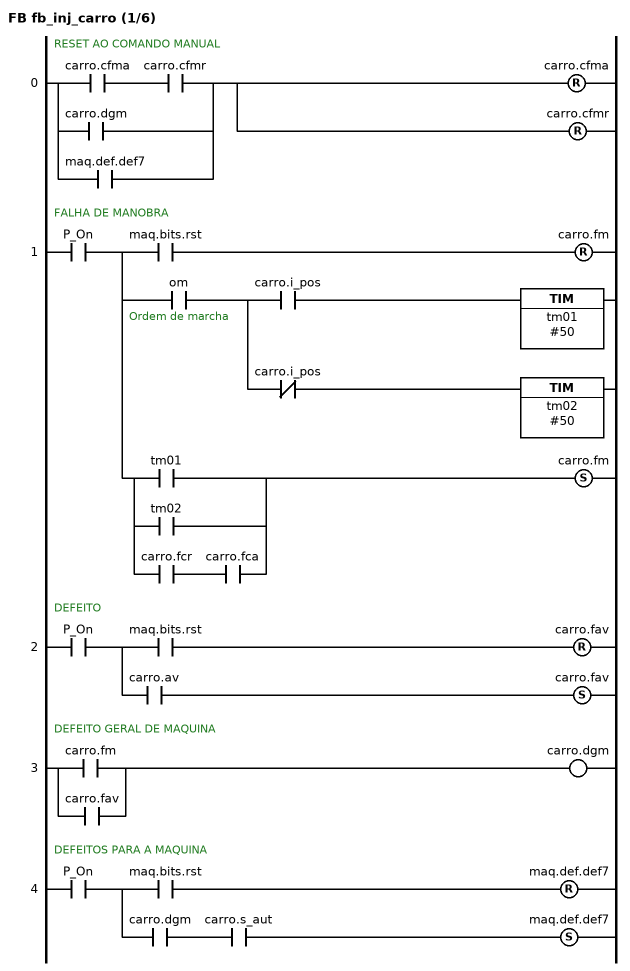
; [picture p48: FB fb_inj_carro, rungs 0-4]
; rung 0: RESET AO COMANDO MANUAL
LD carro.cfma
AND carro.cfmr
OR carro.dgm
OR maq.def.def7
RSET carro.cfma
RSET carro.cfmr
; rung 1: FALHA DE MANOBRA
LD P_On
OUT TR0
AND maq.bits.rst
RSET carro.fm
LD TR0
AND om  ; Ordem de marcha
OUT TR1
AND carro.i_pos
TIM tm01 #50
LD TR1
ANDNOT carro.i_pos
TIM tm02 #50
LD TR0
LD tm01
OR tm02
LD carro.fcr
AND carro.fca
ORLD
ANDLD
SET carro.fm
; rung 2: DEFEITO
LD P_On
OUT TR0
AND maq.bits.rst
RSET carro.fav
LD TR0
AND carro.av
SET carro.fav
; rung 3: DEFEITO GERAL DE MAQUINA
LD carro.fm
OR carro.fav
OUT carro.dgm
; rung 4: DEFEITOS PARA A MAQUINA
LD P_On
OUT TR0
AND maq.bits.rst
RSET maq.def.def7
LD TR0
AND carro.dgm
AND carro.s_aut
SET maq.def.def7

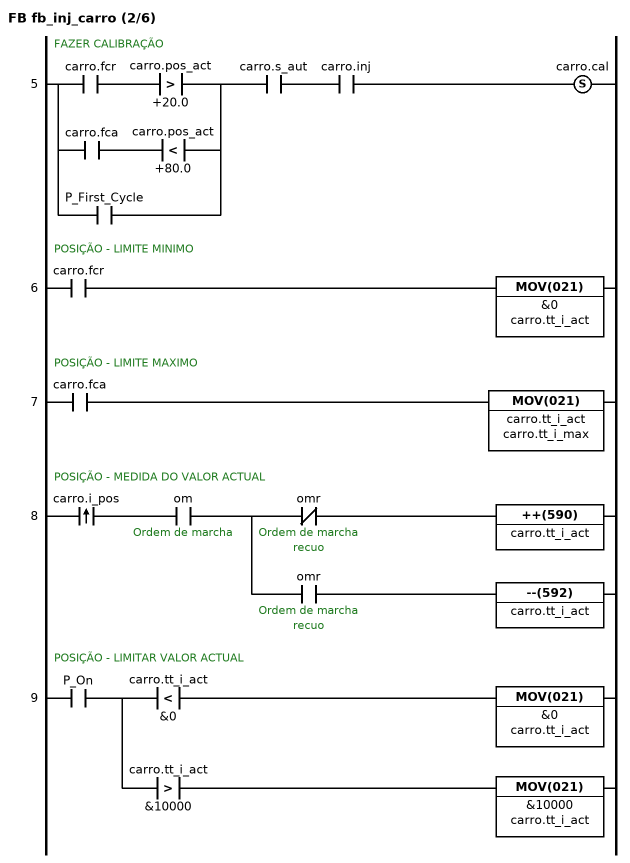
; rung 5: FAZER CALIBRAÇÃO
LD carro.fcr
AND>F(333) carro.pos_act +20.0
LD carro.fca
AND<F(331) carro.pos_act +80.0
ORLD
OR P_First_Cycle
AND carro.s_aut
AND carro.inj
SET carro.cal
; rung 6: POSIÇÃO - LIMITE MINIMO
LD carro.fcr
MOV(021) &0 carro.tt_i_act
; rung 7: POSIÇÃO - LIMITE MAXIMO
LD carro.fca
MOV(021) carro.tt_i_act carro.tt_i_max
; rung 8: POSIÇÃO - MEDIDA DO VALOR ACTUAL
@LD carro.i_pos
AND om  ; Ordem de marcha
OUT TR0
ANDNOT omr  ; Ordem de marcha recuo
++(590) carro.tt_i_act
LD TR0
AND omr  ; Ordem de marcha recuo
--(592) carro.tt_i_act
; rung 9: POSIÇÃO - LIMITAR VALOR ACTUAL
LD P_On
OUT TR0
AND<(310) carro.tt_i_act &0
MOV(021) &0 carro.tt_i_act
LD TR0
AND>(320) carro.tt_i_act &10000
MOV(021) &10000 carro.tt_i_act

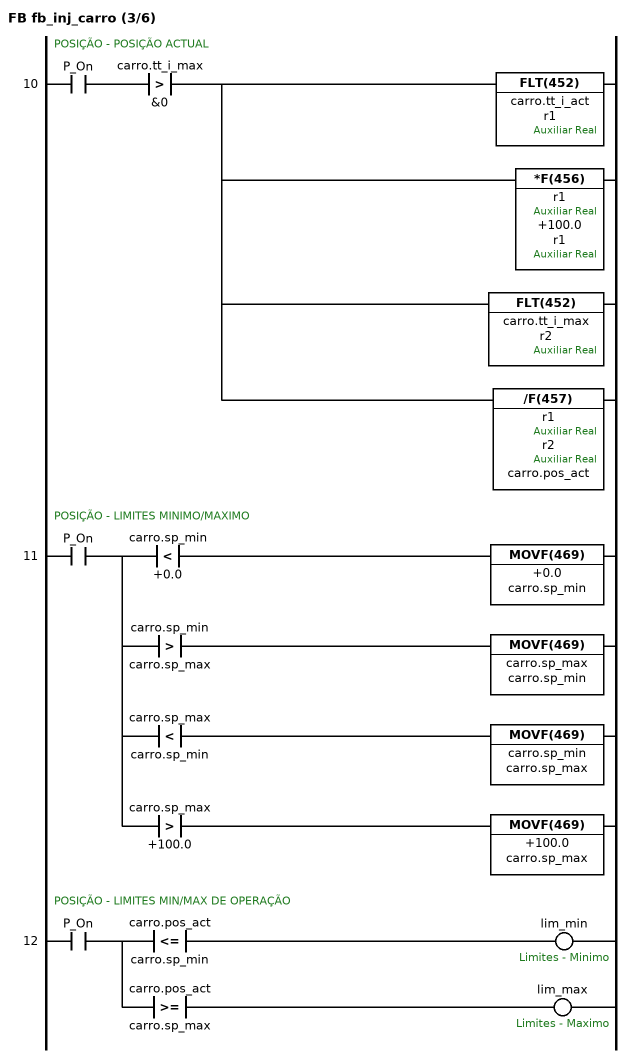
; rung 10: POSIÇÃO - POSIÇÃO ACTUAL
LD P_On
AND>(320) carro.tt_i_max &0
FLT(452) carro.tt_i_act r1  ; Auxiliar Real
*F(456) r1 +100.0 r1  ; Auxiliar Real
FLT(452) carro.tt_i_max r2  ; Auxiliar Real
/F(457) r1 r2 carro.pos_act  ; Auxiliar Real
; rung 11: POSIÇÃO - LIMITES MINIMO/MAXIMO
LD P_On
OUT TR0
AND<F(331) carro.sp_min +0.0
MOVF(469) +0.0 carro.sp_min
LD TR0
AND>F(333) carro.sp_min carro.sp_max
MOVF(469) carro.sp_max carro.sp_min
LD TR0
AND<F(331) carro.sp_max carro.sp_min
MOVF(469) carro.sp_min carro.sp_max
LD TR0
AND>F(333) carro.sp_max +100.0
MOVF(469) +100.0 carro.sp_max
; rung 12: POSIÇÃO - LIMITES MIN/MAX DE OPERAÇÃO
LD P_On
OUT TR0
AND<=F(332) carro.pos_act carro.sp_min
OUT lim_min  ; Limites - Minimo
LD TR0
AND>=F(334) carro.pos_act carro.sp_max
OUT lim_max  ; Limites - Maximo

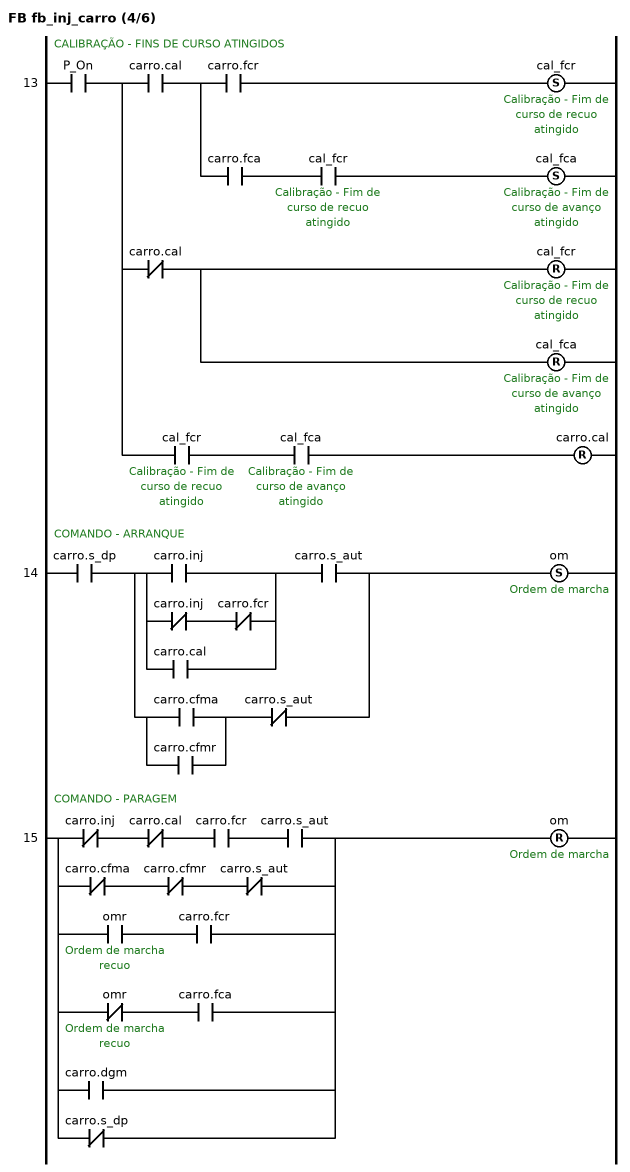
; rung 13: CALIBRAÇÃO - FINS DE CURSO ATINGIDOS
LD P_On
OUT TR0
AND carro.cal
OUT TR1
AND carro.fcr
SET cal_fcr  ; Calibração - Fim de curso de recuo atingido
LD TR1
AND carro.fca
AND cal_fcr  ; Calibração - Fim de curso de recuo atingido
SET cal_fca  ; Calibração - Fim de curso de avanço atingido
LD TR0
ANDNOT carro.cal
RSET cal_fcr  ; Calibração - Fim de curso de recuo atingido
RSET cal_fca  ; Calibração - Fim de curso de avanço atingido
LD TR0
AND cal_fcr  ; Calibração - Fim de curso de recuo atingido
AND cal_fca  ; Calibração - Fim de curso de avanço atingido
RSET carro.cal
; rung 14: COMANDO - ARRANQUE
LD carro.s_dp
LD carro.inj
LDNOT carro.inj
ANDNOT carro.fcr
ORLD
OR carro.cal
AND carro.s_aut
LD carro.cfma
OR carro.cfmr
ANDNOT carro.s_aut
ORLD
ANDLD
SET om  ; Ordem de marcha
; rung 15: COMANDO - PARAGEM
LDNOT carro.inj
ANDNOT carro.cal
AND carro.fcr
AND carro.s_aut
LDNOT carro.cfma
ANDNOT carro.cfmr
ANDNOT carro.s_aut
ORLD
LD omr  ; Ordem de marcha recuo
AND carro.fcr
ORLD
LDNOT omr  ; Ordem de marcha recuo
AND carro.fca
ORLD
OR carro.dgm
ORNOT carro.s_dp
RSET om  ; Ordem de marcha

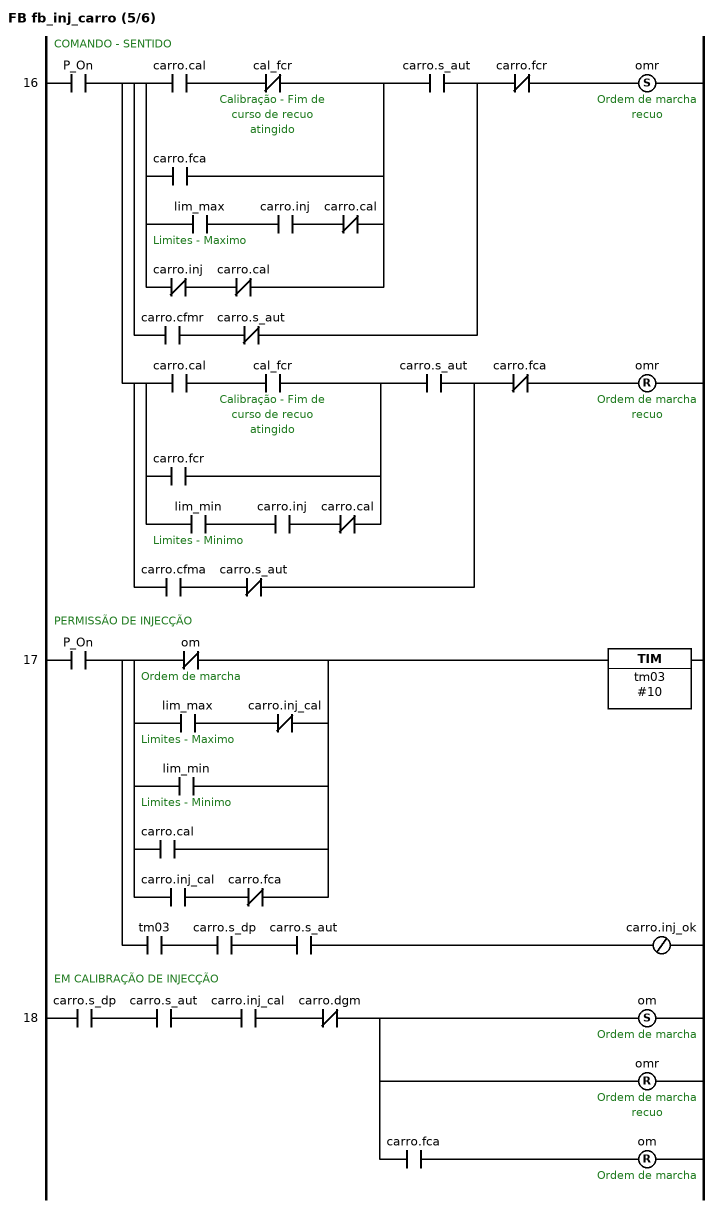
; rung 16: COMANDO - SENTIDO
LD P_On
OUT TR0
LD carro.cal
ANDNOT cal_fcr  ; Calibração - Fim de curso de recuo atingido
OR carro.fca
LD lim_max  ; Limites - Maximo
AND carro.inj
ANDNOT carro.cal
ORLD
LDNOT carro.inj
ANDNOT carro.cal
ORLD
AND carro.s_aut
LD carro.cfmr
ANDNOT carro.s_aut
ORLD
ANDLD
ANDNOT carro.fcr
SET omr  ; Ordem de marcha recuo
LD TR0
LD carro.cal
AND cal_fcr  ; Calibração - Fim de curso de recuo atingido
OR carro.fcr
LD lim_min  ; Limites - Minimo
AND carro.inj
ANDNOT carro.cal
ORLD
AND carro.s_aut
LD carro.cfma
ANDNOT carro.s_aut
ORLD
ANDLD
ANDNOT carro.fca
RSET omr  ; Ordem de marcha recuo
; rung 17: PERMISSÃO DE INJECÇÃO
LD P_On
OUT TR0
LDNOT om  ; Ordem de marcha
LD lim_max  ; Limites - Maximo
ANDNOT carro.inj_cal
ORLD
OR lim_min  ; Limites - Minimo
OR carro.cal
LD carro.inj_cal
ANDNOT carro.fca
ORLD
ANDLD
TIM tm03 #10
LD TR0
AND tm03
AND carro.s_dp
AND carro.s_aut
OUTNOT carro.inj_ok
; rung 18: EM CALIBRAÇÃO DE INJECÇÃO
LD carro.s_dp
AND carro.s_aut
AND carro.inj_cal
ANDNOT carro.dgm
SET om  ; Ordem de marcha
RSET omr  ; Ordem de marcha recuo
AND carro.fca
RSET om  ; Ordem de marcha

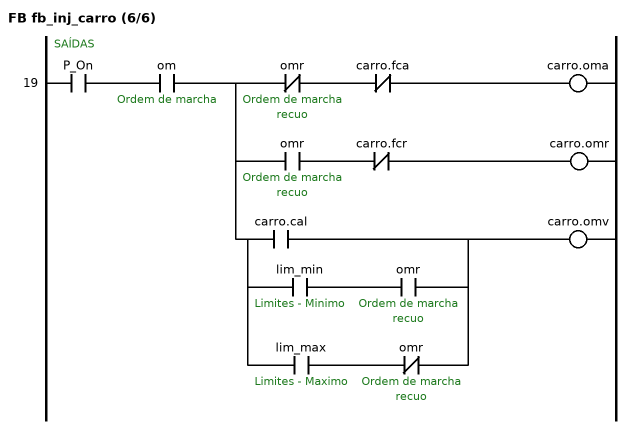
; rung 19: SAÍDAS
LD P_On
AND om  ; Ordem de marcha
OUT TR0
ANDNOT omr  ; Ordem de marcha recuo
ANDNOT carro.fca
OUT carro.oma
LD TR0
AND omr  ; Ordem de marcha recuo
ANDNOT carro.fcr
OUT carro.omr
LD TR0
LD carro.cal
LD lim_min  ; Limites - Minimo
AND omr  ; Ordem de marcha recuo
ORLD
LD lim_max  ; Limites - Maximo
ANDNOT omr  ; Ordem de marcha recuo
ORLD
ANDLD
OUT carro.omv

## Function block fb_inj_caudal
; FUNÇÃO CAUDALIMETRO - Caudalimetro local/remoto
VAR_IN_OUT
  tt : s_caudal;  (* Dados do caudalímetro *)
END_VAR
VAR
  tt_rem_d : REAL;  (* Diferença de totalização *)
  tm01 : TIMER;
  tm02 : TIMER;
  ct01 : COUNTER;
END_VAR

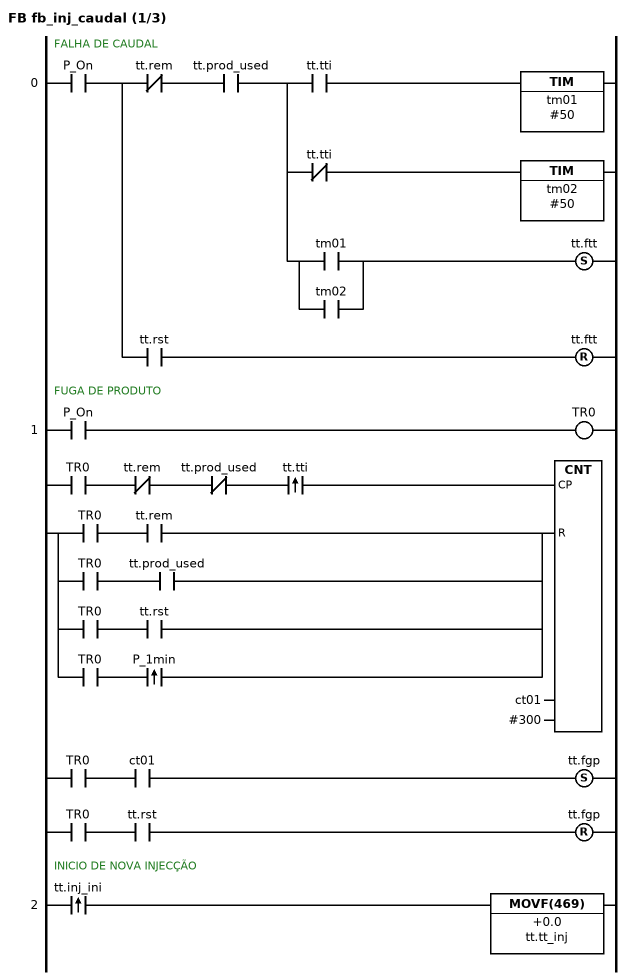
; rung 0: FALHA DE CAUDAL
LD P_On
OUT TR0
ANDNOT tt.rem
AND tt.prod_used
OUT TR1
AND tt.tti
TIM tm01 #50
LD TR1
ANDNOT tt.tti
TIM tm02 #50
LD TR1
LD tm01
OR tm02
ANDLD
SET tt.ftt
LD TR0
AND tt.rst
RSET tt.ftt
; rung 1: FUGA DE PRODUTO
LD P_On
OUT TR0
LD TR0
ANDNOT tt.rem
ANDNOT tt.prod_used
@AND tt.tti
LD TR0
AND tt.rem
LD TR0
AND tt.prod_used
ORLD
LD TR0
AND tt.rst
ORLD
LD TR0
@AND P_1min
ORLD
CNT ct01 #300
LD TR0
AND ct01
SET tt.fgp
LD TR0
AND tt.rst
RSET tt.fgp
; rung 2: INICIO DE NOVA INJECÇÃO
@LD tt.inj_ini
MOVF(469) +0.0 tt.tt_inj

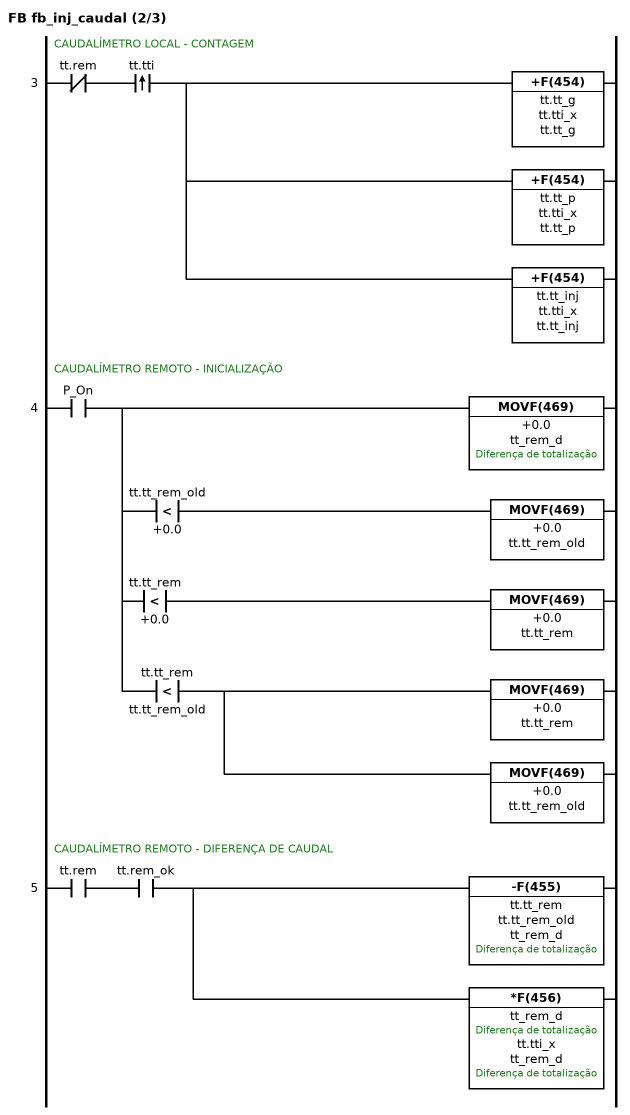
; rung 3: CAUDALÍMETRO LOCAL - CONTAGEM
LDNOT tt.rem
@AND tt.tti
+F(454) tt.tt_g tt.tti_x tt.tt_g
+F(454) tt.tt_p tt.tti_x tt.tt_p
+F(454) tt.tt_inj tt.tti_x tt.tt_inj
; rung 4: CAUDALÍMETRO REMOTO - INICIALIZAÇÃO
LD P_On
OUT TR0
MOVF(469) +0.0 tt_rem_d  ; Diferença de totalização
AND<F(331) tt.tt_rem_old +0.0
MOVF(469) +0.0 tt.tt_rem_old
LD TR0
AND<F(331) tt.tt_rem +0.0
MOVF(469) +0.0 tt.tt_rem
LD TR0
AND<F(331) tt.tt_rem tt.tt_rem_old
MOVF(469) +0.0 tt.tt_rem
MOVF(469) +0.0 tt.tt_rem_old
; rung 5: CAUDALÍMETRO REMOTO - DIFERENÇA DE CAUDAL
LD tt.rem
AND tt.rem_ok
-F(455) tt.tt_rem tt.tt_rem_old tt_rem_d  ; Diferença de totalização
*F(456) tt_rem_d tt.tti_x tt_rem_d  ; Diferença de totalização

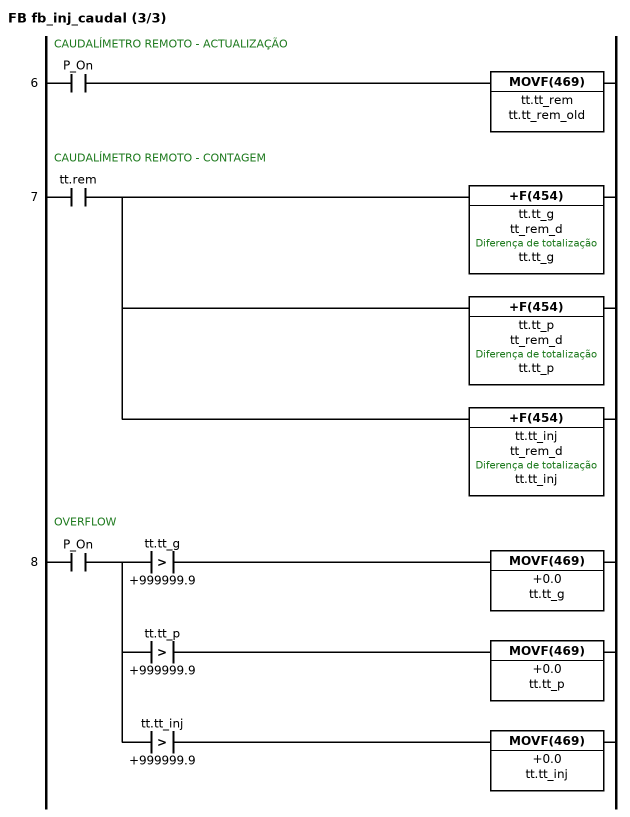
; rung 6: CAUDALÍMETRO REMOTO - ACTUALIZAÇÃO
LD P_On
MOVF(469) tt.tt_rem tt.tt_rem_old
; rung 7: CAUDALÍMETRO REMOTO - CONTAGEM
LD tt.rem
+F(454) tt.tt_g tt_rem_d tt.tt_g  ; Diferença de totalização
+F(454) tt.tt_p tt_rem_d tt.tt_p  ; Diferença de totalização
+F(454) tt.tt_inj tt_rem_d tt.tt_inj  ; Diferença de totalização
; rung 8: OVERFLOW
LD P_On
OUT TR0
AND>F(333) tt.tt_g +999999.9
MOVF(469) +0.0 tt.tt_g
LD TR0
AND>F(333) tt.tt_p +999999.9
MOVF(469) +0.0 tt.tt_p
LD TR0
AND>F(333) tt.tt_inj +999999.9
MOVF(469) +0.0 tt.tt_inj

## Function block fb_maquina
; FUNÇÃO MAQUINA - Faz a gestão dos passos e comandos aos vários blocos.
VAR_INPUT
  Rcp_OK : BOOL;
END_VAR
VAR_IN_OUT
  maq : s_maquina;  (* Dados da maquina *)
  of1_exe : s_of;  (* Dados da OF a ser executada *)
  of2_maq : s_of;  (* Dados da OF carregados na maquina *)
  of3_trp : s_of;  (* Dados da OF recebidos do transporte *)
  mes_com : s_mes_com;  (* Dados da comunição com o MES *)
  prg_exe : s_of_prg;  (* Programa a executar *)
  prg_on : s_of_prg;  (* Programa online *)
  Estado : s_Estado;
  F_Ciclo_bit : BOOL;
END_VAR
VAR
  fb_maquina_mov_pss_act : fb_maquina_mov_pss_act;
  fb_of_copy : fb_of_copy;
  fb_of_clear : fb_of_clear;
  fb_mes_com_exe : fb_mes_com_exe;
  fb_maquina_copy_log : fb_maquina_copy_log;
  fb_of_copy_of_prg_prg : fb_of_copy_of_prg_prg;
  fb_of_exe_calc : fb_of_exe_calc;
  log_tipo : INT;  (* Tipo de copia: 0 - Copia user/lote e dados a zero / 1 - Copia com ordem a decorrer (não copia user/lote) / 2 - Fim da ordem (Coloca passo 999) / 3 - Ordem descarregada sem execução (Colocar -3 no passo) *)
  tm01 : TIMER;
  tm02 : TIMER;
  tm03 : TIMER;
  tm04 : TIMER;
  tm05 : TIMER;
  tm06 : TIMER;
  tm07 : TIMER;
  tm08 : TIMER;
  tm09 : TIMER;
  tm10 : TIMER;
  tm11 : TIMER;
  tm12 : TIMER;
  tm13 : TIMER;
  tm14 : TIMER;
  tm15 : TIMER;
  tm16 : TIMER;
  of_trat : BOOL;  (* Ordem tratada *)
END_VAR

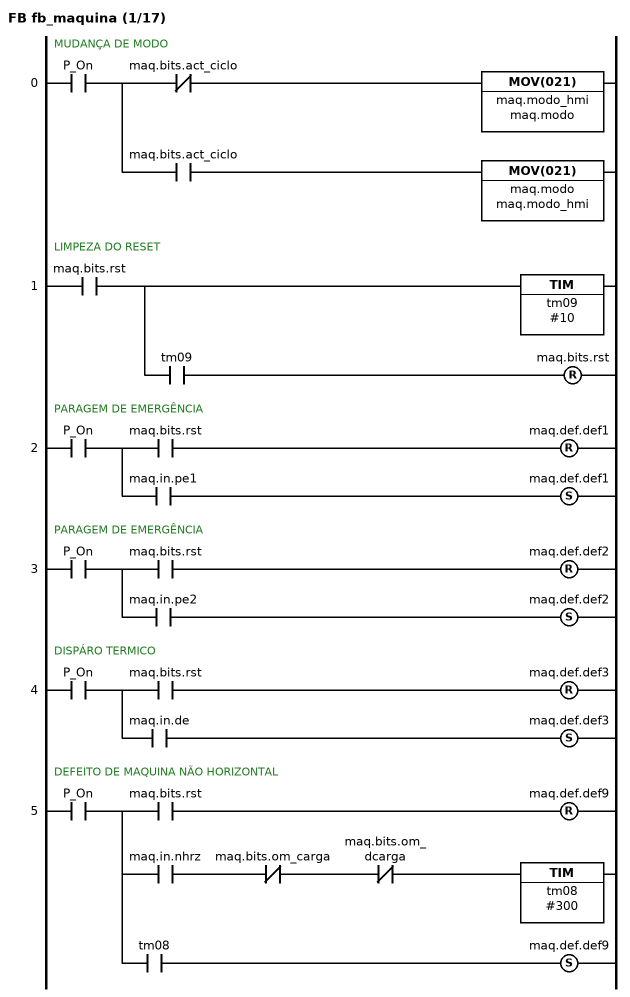
; rung 0: MUDANÇA DE MODO
LD P_On
OUT TR0
ANDNOT maq.bits.act_ciclo
MOV(021) maq.modo_hmi maq.modo
LD TR0
AND maq.bits.act_ciclo
MOV(021) maq.modo maq.modo_hmi
; rung 1: LIMPEZA DO RESET
LD maq.bits.rst
TIM tm09 #10
AND tm09
RSET maq.bits.rst
; rung 2: PARAGEM DE EMERGÊNCIA
LD P_On
OUT TR0
AND maq.bits.rst
RSET maq.def.def1
LD TR0
AND maq.in.pe1
SET maq.def.def1
; rung 3: PARAGEM DE EMERGÊNCIA
LD P_On
OUT TR0
AND maq.bits.rst
RSET maq.def.def2
LD TR0
AND maq.in.pe2
SET maq.def.def2
; rung 4: DISPÁRO TERMICO
LD P_On
OUT TR0
AND maq.bits.rst
RSET maq.def.def3
LD TR0
AND maq.in.de
SET maq.def.def3
; rung 5: DEFEITO DE MAQUINA NÃO HORIZONTAL
LD P_On
OUT TR0
AND maq.bits.rst
RSET maq.def.def9
LD TR0
AND maq.in.nhrz
ANDNOT maq.bits.om_carga
ANDNOT maq.bits.om_dcarga
TIM tm08 #300
LD TR0
AND tm08
SET maq.def.def9

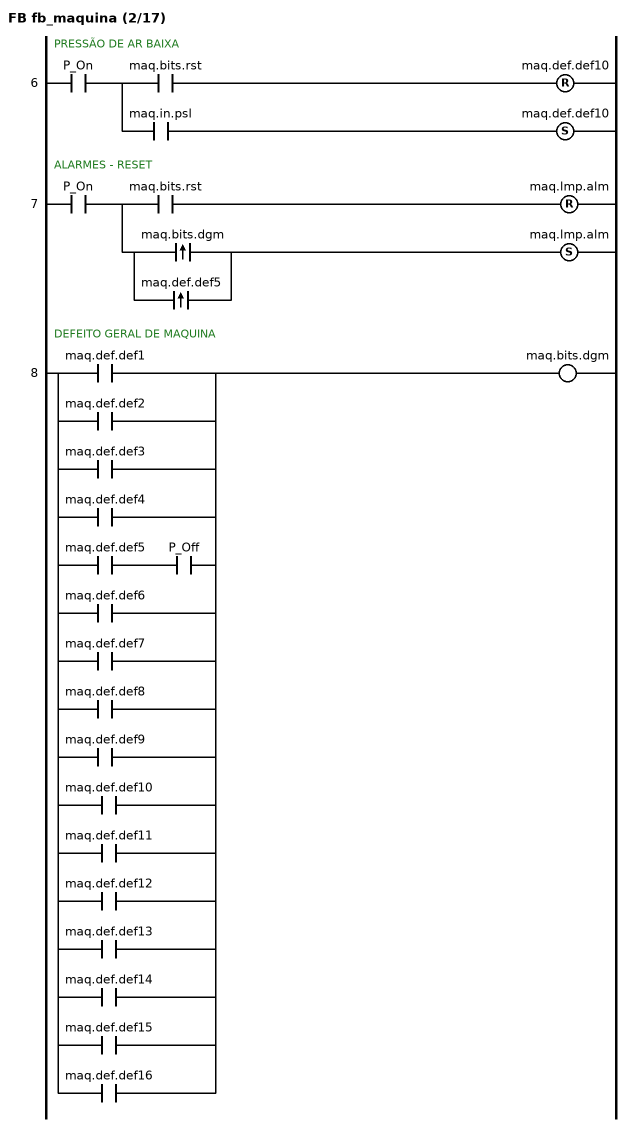
; rung 6: PRESSÃO DE AR BAIXA
LD P_On
OUT TR0
AND maq.bits.rst
RSET maq.def.def10
LD TR0
AND maq.in.psl
SET maq.def.def10
; rung 7: ALARMES - RESET
LD P_On
OUT TR0
AND maq.bits.rst
RSET maq.lmp.alm
LD TR0
@LD maq.bits.dgm
@OR maq.def.def5
ANDLD
SET maq.lmp.alm
; rung 8: DEFEITO GERAL DE MAQUINA
LD maq.def.def1
OR maq.def.def2
OR maq.def.def3
OR maq.def.def4
LD maq.def.def5
AND P_Off
ORLD
OR maq.def.def6
OR maq.def.def7
OR maq.def.def8
OR maq.def.def9
OR maq.def.def10
OR maq.def.def11
OR maq.def.def12
OR maq.def.def13
OR maq.def.def14
OR maq.def.def15
OR maq.def.def16
OUT maq.bits.dgm

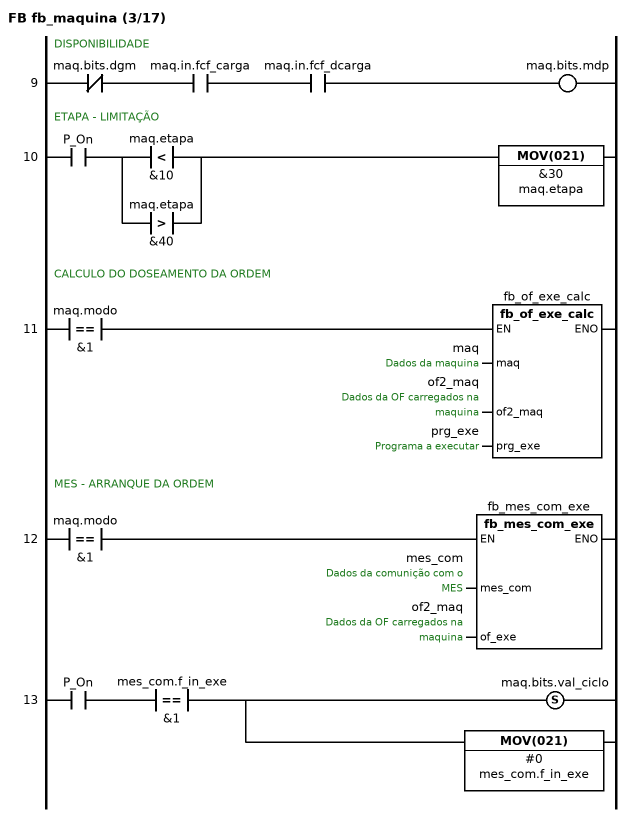
; rung 9: DISPONIBILIDADE
LDNOT maq.bits.dgm
AND maq.in.fcf_carga
AND maq.in.fcf_dcarga
OUT maq.bits.mdp
; rung 10: ETAPA - LIMITAÇÃO
LD P_On
LD<(310) maq.etapa &10
OR>(320) maq.etapa &40
ANDLD
MOV(021) &30 maq.etapa
; rung 11: CALCULO DO DOSEAMENTO DA ORDEM
LD=(300) maq.modo &1
CALL fb_of_exe_calc : fb_of_exe_calc (maq := maq, of2_maq := of2_maq, prg_exe := prg_exe)  ; Dados da maquina, Dados da OF carregados na maquina, Programa a executar
; rung 12: MES - ARRANQUE DA ORDEM
LD=(300) maq.modo &1
CALL fb_mes_com_exe : fb_mes_com_exe (mes_com := mes_com, of_exe := of2_maq)  ; Dados da comunição com o MES, Dados da OF carregados na maquina
; rung 13
LD P_On
AND=(300) mes_com.f_in_exe &1
SET maq.bits.val_ciclo
MOV(021) #0 mes_com.f_in_exe

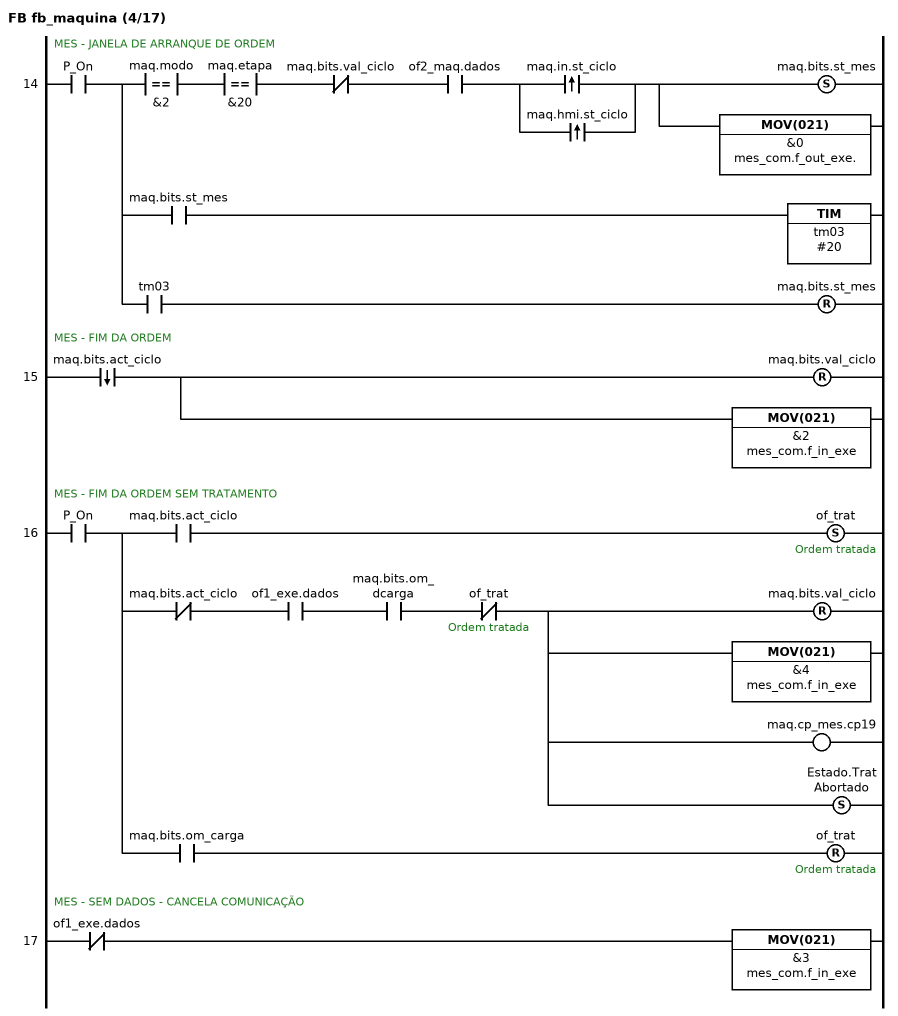
; rung 14: MES - JANELA DE ARRANQUE DE ORDEM
LD P_On
OUT TR0
AND=(300) maq.modo &2
AND=(300) maq.etapa &20
ANDNOT maq.bits.val_ciclo
AND of2_maq.dados
@LD maq.in.st_ciclo
@OR maq.hmi.st_ciclo
ANDLD
SET maq.bits.st_mes
MOV(021) &0 mes_com.f_out_exe.
LD TR0
AND maq.bits.st_mes
TIM tm03 #20
LD TR0
AND tm03
RSET maq.bits.st_mes
; rung 15: MES - FIM DA ORDEM
%LD maq.bits.act_ciclo
RSET maq.bits.val_ciclo
MOV(021) &2 mes_com.f_in_exe
; rung 16: MES - FIM DA ORDEM SEM TRATAMENTO
LD P_On
OUT TR0
AND maq.bits.act_ciclo
SET of_trat  ; Ordem tratada
LD TR0
ANDNOT maq.bits.act_ciclo
AND of1_exe.dados
AND maq.bits.om_dcarga
ANDNOT of_trat  ; Ordem tratada
RSET maq.bits.val_ciclo
MOV(021) &4 mes_com.f_in_exe
OUT maq.cp_mes.cp19
SET Estado.TratAbortado
LD TR0
AND maq.bits.om_carga
RSET of_trat  ; Ordem tratada
; rung 17: MES - SEM DADOS - CANCELA COMUNICAÇÃO
LDNOT of1_exe.dados
MOV(021) &3 mes_com.f_in_exe

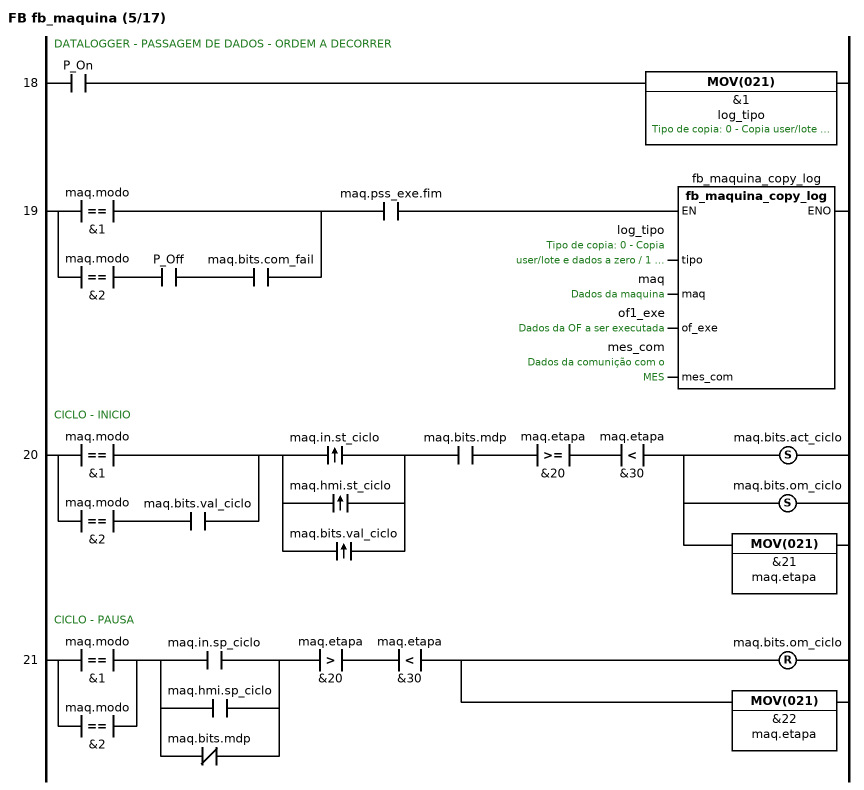
; rung 18: DATALOGGER - PASSAGEM DE DADOS - ORDEM A DECORRER
LD P_On
MOV(021) &1 log_tipo  ; Tipo de copia: 0 - Copia user/lote e dados a zero / 1 - Copia com ordem a decorrer (não copia user/lote) / 2 - Fim da ordem (Coloca passo 999) / 3 - Ordem descarregada sem execução (Colocar -3 no passo)
; rung 19
LD=(300) maq.modo &1
LD=(300) maq.modo &2
AND P_Off
AND maq.bits.com_fail
ORLD
AND maq.pss_exe.fim
CALL fb_maquina_copy_log : fb_maquina_copy_log (tipo := log_tipo, maq := maq, of_exe := of1_exe, mes_com := mes_com)  ; Tipo de copia: 0 - Copia user/lote e dados a zero / 1 - Copia com ordem a decorrer (não copia user/lote) / 2 - Fim da ordem (Coloca passo 999) / 3 - Ordem descarregada sem execução (Colocar -3 no passo), Dados da maquina, Dados da OF a ser executada, Dados da comunição com o MES
; rung 20: CICLO - INICIO
LD=(300) maq.modo &1
LD=(300) maq.modo &2
AND maq.bits.val_ciclo
ORLD
@LD maq.in.st_ciclo
@OR maq.hmi.st_ciclo
@OR maq.bits.val_ciclo
ANDLD
AND maq.bits.mdp
AND>=(325) maq.etapa &20
AND<(310) maq.etapa &30
SET maq.bits.act_ciclo
SET maq.bits.om_ciclo
MOV(021) &21 maq.etapa
; rung 21: CICLO - PAUSA
LD=(300) maq.modo &1
OR=(300) maq.modo &2
LD maq.in.sp_ciclo
OR maq.hmi.sp_ciclo
ORNOT maq.bits.mdp
ANDLD
AND>(320) maq.etapa &20
AND<(310) maq.etapa &30
RSET maq.bits.om_ciclo
MOV(021) &22 maq.etapa

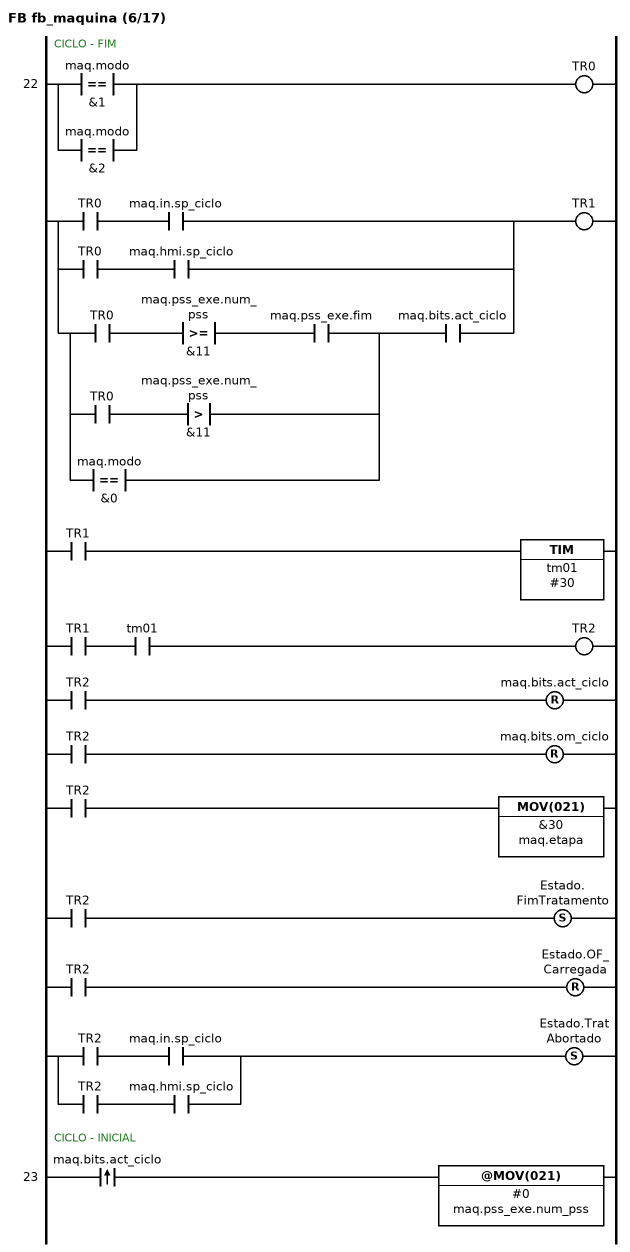
; rung 22: CICLO - FIM
LD=(300) maq.modo &1
OR=(300) maq.modo &2
OUT TR0
LD TR0
AND maq.in.sp_ciclo
LD TR0
AND maq.hmi.sp_ciclo
ORLD
LD TR0
AND>=(325) maq.pss_exe.num_pss &11
AND maq.pss_exe.fim
LD TR0
AND>(320) maq.pss_exe.num_pss &11
ORLD
OR=(300) maq.modo &0
AND maq.bits.act_ciclo
ORLD
OUT TR1
LD TR1
TIM tm01 #30
LD TR1
AND tm01
OUT TR2
LD TR2
RSET maq.bits.act_ciclo
LD TR2
RSET maq.bits.om_ciclo
LD TR2
MOV(021) &30 maq.etapa
LD TR2
SET Estado.FimTratamento
LD TR2
RSET Estado.OF_Carregada
LD TR2
AND maq.in.sp_ciclo
LD TR2
AND maq.hmi.sp_ciclo
ORLD
SET Estado.TratAbortado
; rung 23: CICLO - INICIAL
@LD maq.bits.act_ciclo
@MOV(021) #0 maq.pss_exe.num_pss

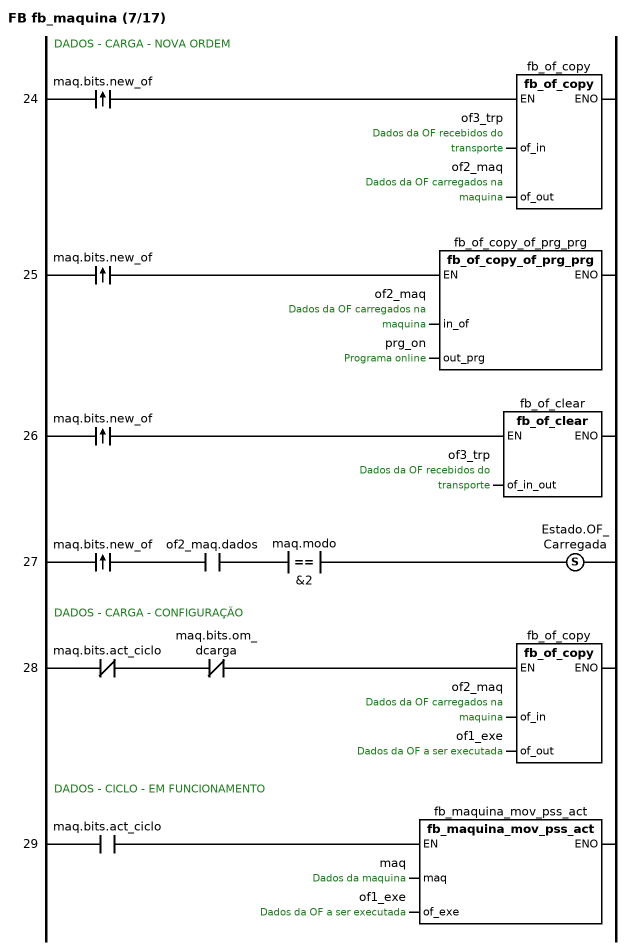
; rung 24: DADOS - CARGA - NOVA ORDEM
@LD maq.bits.new_of
CALL fb_of_copy : fb_of_copy (of_in := of3_trp, of_out := of2_maq)  ; Dados da OF recebidos do transporte, Dados da OF carregados na maquina
; rung 25
@LD maq.bits.new_of
CALL fb_of_copy_of_prg_prg : fb_of_copy_of_prg_prg (in_of := of2_maq, out_prg := prg_on)  ; Dados da OF carregados na maquina, Programa online
; rung 26
@LD maq.bits.new_of
CALL fb_of_clear : fb_of_clear (of_in_out := of3_trp)  ; Dados da OF recebidos do transporte
; rung 27
@LD maq.bits.new_of
AND of2_maq.dados
AND=(300) maq.modo &2
SET Estado.OF_Carregada
; rung 28: DADOS - CARGA - CONFIGURAÇÃO
LDNOT maq.bits.act_ciclo
ANDNOT maq.bits.om_dcarga
CALL fb_of_copy : fb_of_copy (of_in := of2_maq, of_out := of1_exe)  ; Dados da OF carregados na maquina, Dados da OF a ser executada
; rung 29: DADOS - CICLO - EM FUNCIONAMENTO
LD maq.bits.act_ciclo
CALL fb_maquina_mov_pss_act : fb_maquina_mov_pss_act (maq := maq, of_exe := of1_exe)  ; Dados da maquina, Dados da OF a ser executada

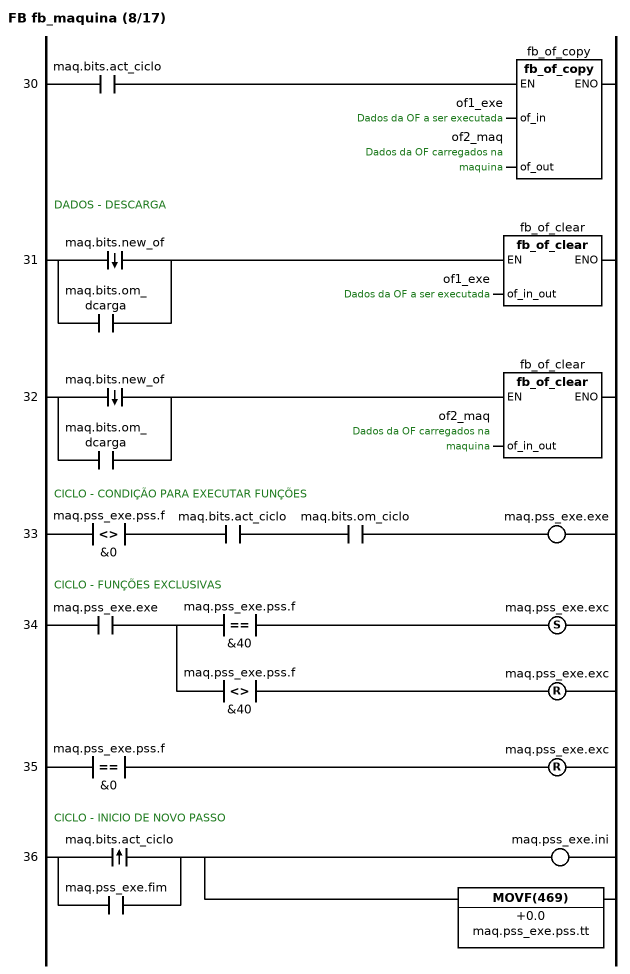
; rung 30
LD maq.bits.act_ciclo
CALL fb_of_copy : fb_of_copy (of_in := of1_exe, of_out := of2_maq)  ; Dados da OF a ser executada, Dados da OF carregados na maquina
; rung 31: DADOS - DESCARGA
%LD maq.bits.new_of
OR maq.bits.om_dcarga
CALL fb_of_clear : fb_of_clear (of_in_out := of1_exe)  ; Dados da OF a ser executada
; rung 32
%LD maq.bits.new_of
OR maq.bits.om_dcarga
CALL fb_of_clear : fb_of_clear (of_in_out := of2_maq)  ; Dados da OF carregados na maquina
; rung 33: CICLO - CONDIÇÃO PARA EXECUTAR FUNÇÕES
LD<>(305) maq.pss_exe.pss.f &0
AND maq.bits.act_ciclo
AND maq.bits.om_ciclo
OUT maq.pss_exe.exe
; rung 34: CICLO - FUNÇÕES EXCLUSIVAS
LD maq.pss_exe.exe
OUT TR0
AND=(300) maq.pss_exe.pss.f &40
SET maq.pss_exe.exc
LD TR0
AND<>(305) maq.pss_exe.pss.f &40
RSET maq.pss_exe.exc
; rung 35
LD=(300) maq.pss_exe.pss.f &0
RSET maq.pss_exe.exc
; rung 36: CICLO - INICIO DE NOVO PASSO
@LD maq.bits.act_ciclo
OR maq.pss_exe.fim
OUT maq.pss_exe.ini
MOVF(469) +0.0 maq.pss_exe.pss.tt

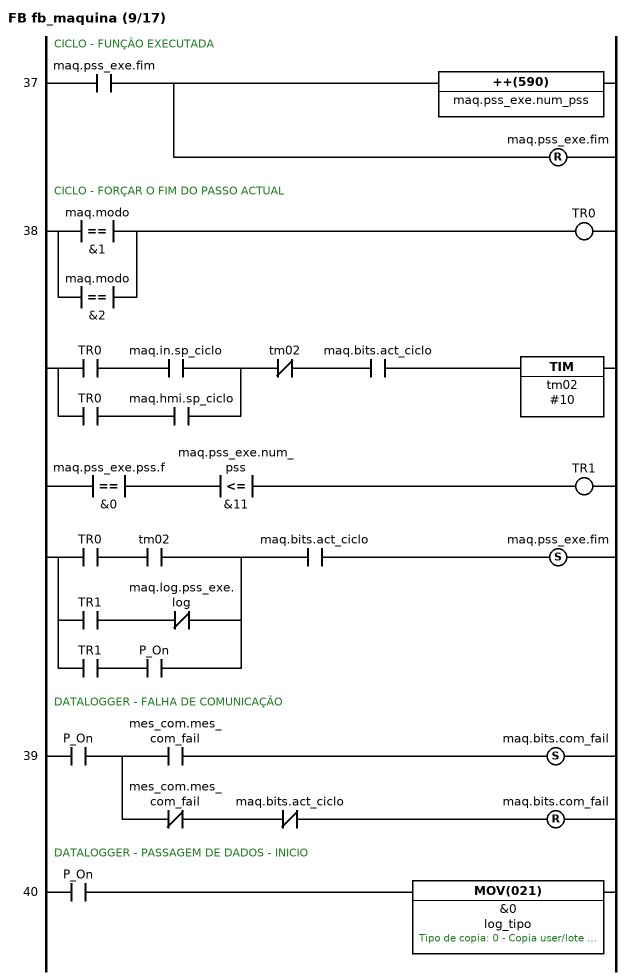
; rung 37: CICLO - FUNÇÃO EXECUTADA
LD maq.pss_exe.fim
++(590) maq.pss_exe.num_pss
RSET maq.pss_exe.fim
; rung 38: CICLO - FORÇAR O FIM DO PASSO ACTUAL
LD=(300) maq.modo &1
OR=(300) maq.modo &2
OUT TR0
LD TR0
AND maq.in.sp_ciclo
LD TR0
AND maq.hmi.sp_ciclo
ORLD
ANDNOT tm02
AND maq.bits.act_ciclo
TIM tm02 #10
LD=(300) maq.pss_exe.pss.f &0
AND<=(315) maq.pss_exe.num_pss &11
OUT TR1
LD TR0
AND tm02
LD TR1
ANDNOT maq.log.pss_exe.log
ORLD
LD TR1
AND P_On
ORLD
AND maq.bits.act_ciclo
SET maq.pss_exe.fim
; rung 39: DATALOGGER - FALHA DE COMUNICAÇÃO
LD P_On
OUT TR0
AND mes_com.mes_com_fail
SET maq.bits.com_fail
LD TR0
ANDNOT mes_com.mes_com_fail
ANDNOT maq.bits.act_ciclo
RSET maq.bits.com_fail
; rung 40: DATALOGGER - PASSAGEM DE DADOS - INICIO
LD P_On
MOV(021) &0 log_tipo  ; Tipo de copia: 0 - Copia user/lote e dados a zero / 1 - Copia com ordem a decorrer (não copia user/lote) / 2 - Fim da ordem (Coloca passo 999) / 3 - Ordem descarregada sem execução (Colocar -3 no passo)

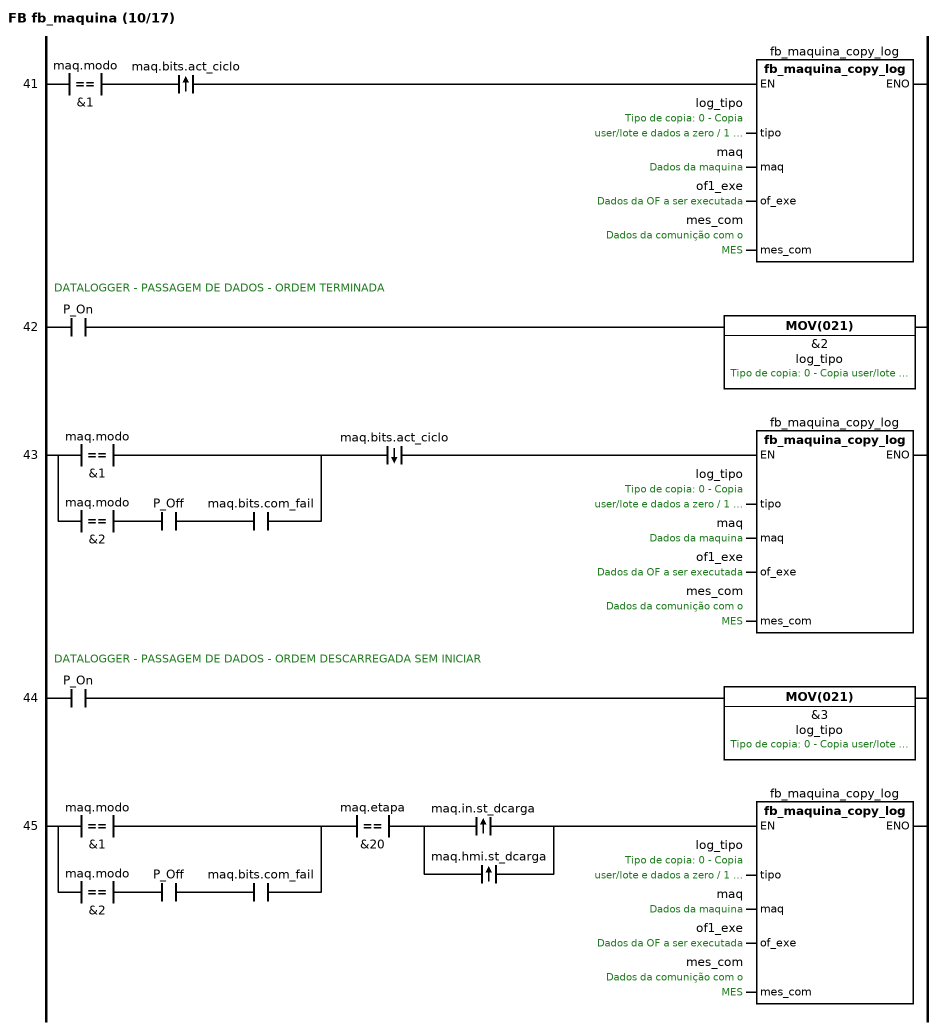
; rung 41
LD=(300) maq.modo &1
@AND maq.bits.act_ciclo
CALL fb_maquina_copy_log : fb_maquina_copy_log (tipo := log_tipo, maq := maq, of_exe := of1_exe, mes_com := mes_com)  ; Tipo de copia: 0 - Copia user/lote e dados a zero / 1 - Copia com ordem a decorrer (não copia user/lote) / 2 - Fim da ordem (Coloca passo 999) / 3 - Ordem descarregada sem execução (Colocar -3 no passo), Dados da maquina, Dados da OF a ser executada, Dados da comunição com o MES
; rung 42: DATALOGGER - PASSAGEM DE DADOS - ORDEM TERMINADA
LD P_On
MOV(021) &2 log_tipo  ; Tipo de copia: 0 - Copia user/lote e dados a zero / 1 - Copia com ordem a decorrer (não copia user/lote) / 2 - Fim da ordem (Coloca passo 999) / 3 - Ordem descarregada sem execução (Colocar -3 no passo)
; rung 43
LD=(300) maq.modo &1
LD=(300) maq.modo &2
AND P_Off
AND maq.bits.com_fail
ORLD
%AND maq.bits.act_ciclo
CALL fb_maquina_copy_log : fb_maquina_copy_log (tipo := log_tipo, maq := maq, of_exe := of1_exe, mes_com := mes_com)  ; Tipo de copia: 0 - Copia user/lote e dados a zero / 1 - Copia com ordem a decorrer (não copia user/lote) / 2 - Fim da ordem (Coloca passo 999) / 3 - Ordem descarregada sem execução (Colocar -3 no passo), Dados da maquina, Dados da OF a ser executada, Dados da comunição com o MES
; rung 44: DATALOGGER - PASSAGEM DE DADOS - ORDEM DESCARREGADA SEM INICIAR
LD P_On
MOV(021) &3 log_tipo  ; Tipo de copia: 0 - Copia user/lote e dados a zero / 1 - Copia com ordem a decorrer (não copia user/lote) / 2 - Fim da ordem (Coloca passo 999) / 3 - Ordem descarregada sem execução (Colocar -3 no passo)
; rung 45
LD=(300) maq.modo &1
LD=(300) maq.modo &2
AND P_Off
AND maq.bits.com_fail
ORLD
AND=(300) maq.etapa &20
@LD maq.in.st_dcarga
@OR maq.hmi.st_dcarga
ANDLD
CALL fb_maquina_copy_log : fb_maquina_copy_log (tipo := log_tipo, maq := maq, of_exe := of1_exe, mes_com := mes_com)  ; Tipo de copia: 0 - Copia user/lote e dados a zero / 1 - Copia com ordem a decorrer (não copia user/lote) / 2 - Fim da ordem (Coloca passo 999) / 3 - Ordem descarregada sem execução (Colocar -3 no passo), Dados da maquina, Dados da OF a ser executada, Dados da comunição com o MES

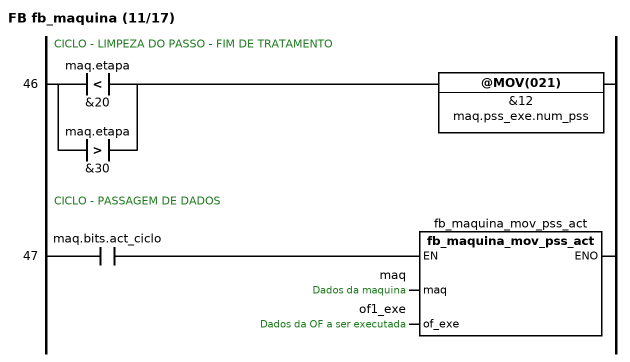
; rung 46: CICLO - LIMPEZA DO PASSO - FIM DE TRATAMENTO
LD<(310) maq.etapa &20
OR>(320) maq.etapa &30
@MOV(021) &12 maq.pss_exe.num_pss
; rung 47: CICLO - PASSAGEM DE DADOS
LD maq.bits.act_ciclo
CALL fb_maquina_mov_pss_act : fb_maquina_mov_pss_act (maq := maq, of_exe := of1_exe)  ; Dados da maquina, Dados da OF a ser executada

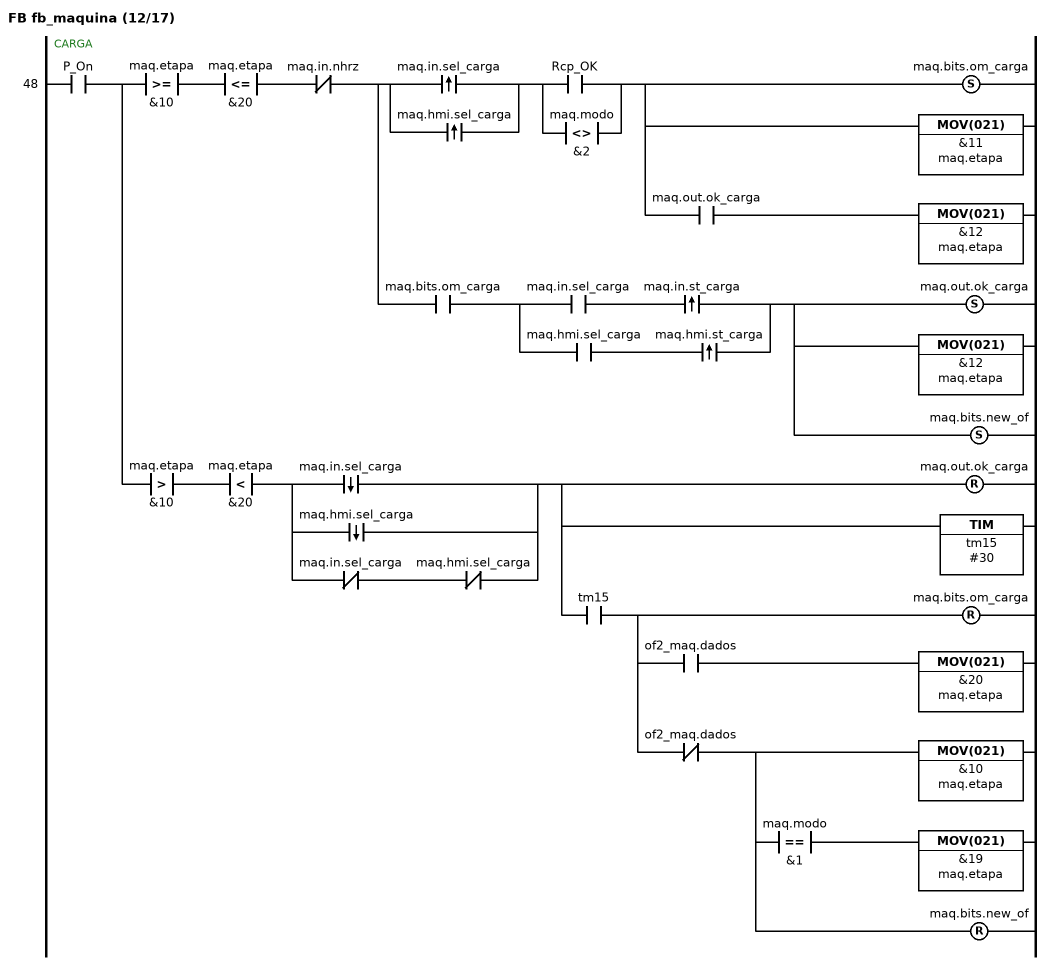
; rung 48: CARGA
LD P_On
OUT TR0
AND>=(325) maq.etapa &10
AND<=(315) maq.etapa &20
ANDNOT maq.in.nhrz
OUT TR1
@LD maq.in.sel_carga
@OR maq.hmi.sel_carga
ANDLD
LD Rcp_OK
OR<>(305) maq.modo &2
ANDLD
SET maq.bits.om_carga
MOV(021) &11 maq.etapa
AND maq.out.ok_carga
MOV(021) &12 maq.etapa
LD TR1
AND maq.bits.om_carga
LD maq.in.sel_carga
@AND maq.in.st_carga
LD maq.hmi.sel_carga
@AND maq.hmi.st_carga
ORLD
ANDLD
SET maq.out.ok_carga
MOV(021) &12 maq.etapa
SET maq.bits.new_of
LD TR0
AND>(320) maq.etapa &10
AND<(310) maq.etapa &20
%LD maq.in.sel_carga
%OR maq.hmi.sel_carga
LDNOT maq.in.sel_carga
ANDNOT maq.hmi.sel_carga
ORLD
ANDLD
RSET maq.out.ok_carga
TIM tm15 #30
AND tm15
OUT TR2
RSET maq.bits.om_carga
AND of2_maq.dados
MOV(021) &20 maq.etapa
LD TR2
ANDNOT of2_maq.dados
OUT TR3
MOV(021) &10 maq.etapa
AND=(300) maq.modo &1
MOV(021) &19 maq.etapa
LD TR3
RSET maq.bits.new_of

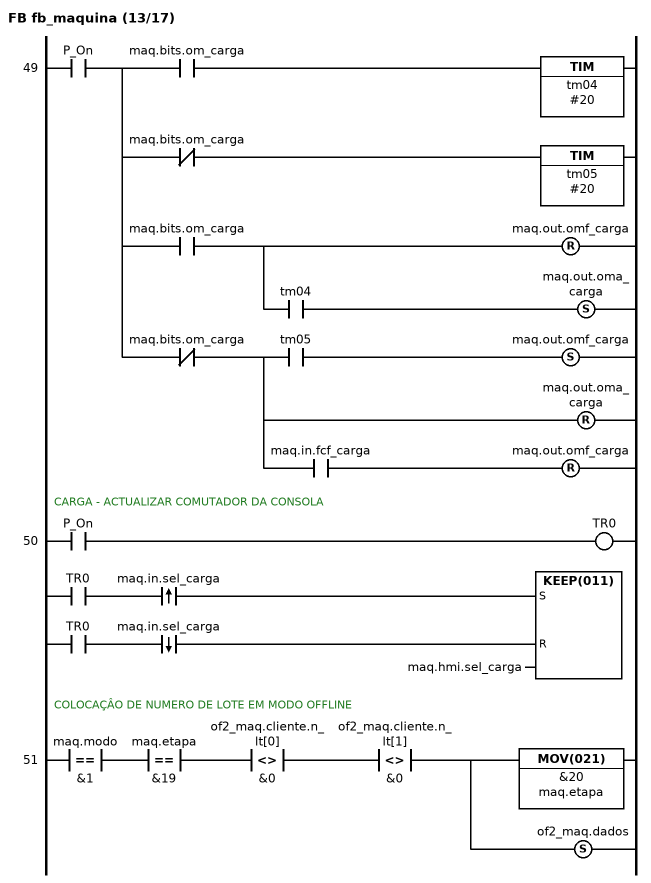
; rung 49
LD P_On
OUT TR0
AND maq.bits.om_carga
TIM tm04 #20
LD TR0
ANDNOT maq.bits.om_carga
TIM tm05 #20
LD TR0
AND maq.bits.om_carga
RSET maq.out.omf_carga
AND tm04
SET maq.out.oma_carga
LD TR0
ANDNOT maq.bits.om_carga
OUT TR1
AND tm05
SET maq.out.omf_carga
LD TR1
RSET maq.out.oma_carga
AND maq.in.fcf_carga
RSET maq.out.omf_carga
; rung 50: CARGA - ACTUALIZAR COMUTADOR DA CONSOLA
LD P_On
OUT TR0
LD TR0
@AND maq.in.sel_carga
LD TR0
%AND maq.in.sel_carga
KEEP(011) maq.hmi.sel_carga
; rung 51: COLOCAÇÂO DE NUMERO DE LOTE EM MODO OFFLINE
LD=(300) maq.modo &1
AND=(300) maq.etapa &19
AND<>(305) of2_maq.cliente.n_lt[0] &0
AND<>(305) of2_maq.cliente.n_lt[1] &0
MOV(021) &20 maq.etapa
SET of2_maq.dados

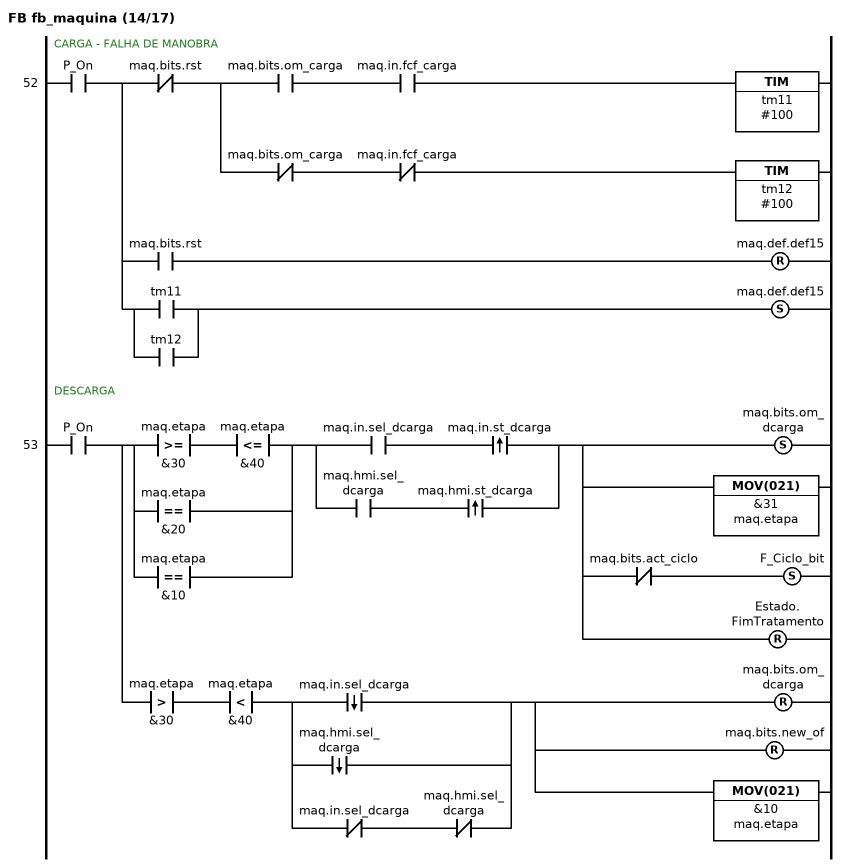
; rung 52: CARGA - FALHA DE MANOBRA
LD P_On
OUT TR0
ANDNOT maq.bits.rst
OUT TR1
AND maq.bits.om_carga
AND maq.in.fcf_carga
TIM tm11 #100
LD TR1
ANDNOT maq.bits.om_carga
ANDNOT maq.in.fcf_carga
TIM tm12 #100
LD TR0
AND maq.bits.rst
RSET maq.def.def15
LD TR0
LD tm11
OR tm12
ANDLD
SET maq.def.def15
; rung 53: DESCARGA
LD P_On
OUT TR0
LD>=(325) maq.etapa &30
AND<=(315) maq.etapa &40
OR=(300) maq.etapa &20
OR=(300) maq.etapa &10
ANDLD
LD maq.in.sel_dcarga
@AND maq.in.st_dcarga
LD maq.hmi.sel_dcarga
@AND maq.hmi.st_dcarga
ORLD
ANDLD
OUT TR1
SET maq.bits.om_dcarga
MOV(021) &31 maq.etapa
ANDNOT maq.bits.act_ciclo
SET F_Ciclo_bit
LD TR1
RSET Estado.FimTratamento
LD TR0
AND>(320) maq.etapa &30
AND<(310) maq.etapa &40
%LD maq.in.sel_dcarga
%OR maq.hmi.sel_dcarga
LDNOT maq.in.sel_dcarga
ANDNOT maq.hmi.sel_dcarga
ORLD
ANDLD
RSET maq.bits.om_dcarga
RSET maq.bits.new_of
MOV(021) &10 maq.etapa

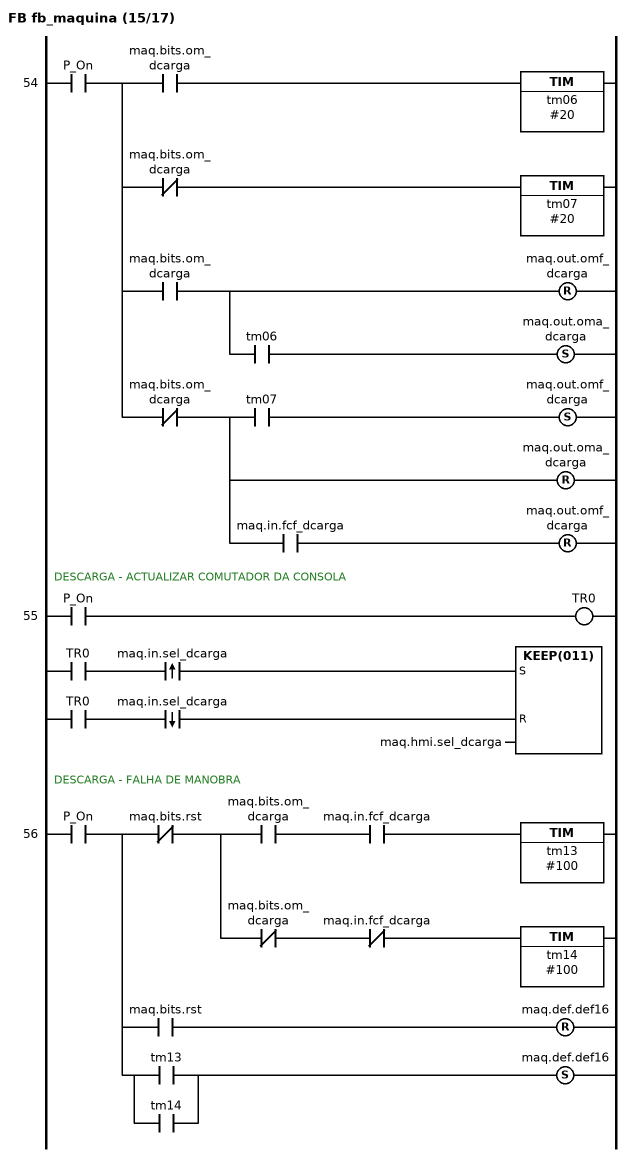
; rung 54
LD P_On
OUT TR0
AND maq.bits.om_dcarga
TIM tm06 #20
LD TR0
ANDNOT maq.bits.om_dcarga
TIM tm07 #20
LD TR0
AND maq.bits.om_dcarga
RSET maq.out.omf_dcarga
AND tm06
SET maq.out.oma_dcarga
LD TR0
ANDNOT maq.bits.om_dcarga
OUT TR1
AND tm07
SET maq.out.omf_dcarga
LD TR1
RSET maq.out.oma_dcarga
AND maq.in.fcf_dcarga
RSET maq.out.omf_dcarga
; rung 55: DESCARGA - ACTUALIZAR COMUTADOR DA CONSOLA
LD P_On
OUT TR0
LD TR0
@AND maq.in.sel_dcarga
LD TR0
%AND maq.in.sel_dcarga
KEEP(011) maq.hmi.sel_dcarga
; rung 56: DESCARGA - FALHA DE MANOBRA
LD P_On
OUT TR0
ANDNOT maq.bits.rst
OUT TR1
AND maq.bits.om_dcarga
AND maq.in.fcf_dcarga
TIM tm13 #100
LD TR1
ANDNOT maq.bits.om_dcarga
ANDNOT maq.in.fcf_dcarga
TIM tm14 #100
LD TR0
AND maq.bits.rst
RSET maq.def.def16
LD TR0
LD tm13
OR tm14
ANDLD
SET maq.def.def16

